(* IEC 61131-3 sources: volt/packages/volt-lsp-iec/test-corpus/lenze-mid/Device/Plc Logic/Application/Library Manager/(unresolved)/cmpopcuastack interfaces (part 3) *)

(* ---- OPCUA_NODEREFERENCE.dut ---- *)
TYPE OPCUA_NODEREFERENCE :
STRUCT
	NODEID : OpcUa_NodeId;
	REFERENCETYPEID : OpcUa_NodeId;
	ISFORWARD : OpcUa_Boolean;
	NOOFREFERENCEDNODEIDS : OpcUa_Int32;
	REFERENCEDNODEIDS : POINTER TO OpcUa_NodeId;
END_STRUCT
END_TYPE

(* ---- OPCUA_NODETYPEDESCRIPTION.dut ---- *)
TYPE OPCUA_NODETYPEDESCRIPTION :
STRUCT
	TYPEDEFINITIONNODE : OpcUa_ExpandedNodeId;
	INCLUDESUBTYPES : OpcUa_Boolean;
	NOOFDATATORETURN : OpcUa_Int32;
	DATATORETURN : POINTER TO OpcUa_QueryDataDescription;
END_STRUCT
END_TYPE

(* ---- OPCUA_NOTIFICATIONMESSAGE.dut ---- *)
TYPE OPCUA_NOTIFICATIONMESSAGE :
STRUCT
	SEQUENCENUMBER : OpcUa_UInt32;
	PUBLISHTIME : OpcUa_DateTime;
	NOOFNOTIFICATIONDATA : OpcUa_Int32;
	NOTIFICATIONDATA : POINTER TO OpcUa_ExtensionObject;
END_STRUCT
END_TYPE

(* ---- OPCUA_OBJECTATTRIBUTES.dut ---- *)
TYPE OPCUA_OBJECTATTRIBUTES :
STRUCT
	SPECIFIEDATTRIBUTES : OpcUa_UInt32;
	DISPLAYNAME : OpcUa_LocalizedText;
	DESCRIPTION : OpcUa_LocalizedText;
	WRITEMASK : OpcUa_UInt32;
	USERWRITEMASK : OpcUa_UInt32;
	EVENTNOTIFIER : OpcUa_Byte;
END_STRUCT
END_TYPE

(* ---- OPCUA_OBJECTTYPEATTRIBUTES.dut ---- *)
TYPE OPCUA_OBJECTTYPEATTRIBUTES :
STRUCT
	SPECIFIEDATTRIBUTES : OpcUa_UInt32;
	DISPLAYNAME : OpcUa_LocalizedText;
	DESCRIPTION : OpcUa_LocalizedText;
	WRITEMASK : OpcUa_UInt32;
	USERWRITEMASK : OpcUa_UInt32;
	ISABSTRACT : OpcUa_Boolean;
END_STRUCT
END_TYPE

(* ---- OPCUA_OPENSECURECHANNELREQUEST.dut ---- *)
TYPE OPCUA_OPENSECURECHANNELREQUEST :
STRUCT
	REQUESTHEADER : OpcUa_RequestHeader;
	CLIENTPROTOCOLVERSION : OpcUa_UInt32;
	REQUESTTYPE : OpcUa_SecurityTokenRequestType;
	SECURITYMODE : OpcUa_MessageSecurityMode;
	CLIENTNONCE : OpcUa_ByteString;
	REQUESTEDLIFETIME : OpcUa_UInt32;
END_STRUCT
END_TYPE

(* ---- OPCUA_OPENSECURECHANNELRESPONSE.dut ---- *)
TYPE OPCUA_OPENSECURECHANNELRESPONSE :
STRUCT
	RESPONSEHEADER : OpcUa_ResponseHeader;
	SERVERPROTOCOLVERSION : OpcUa_UInt32;
	SECURITYTOKEN : OpcUa_ChannelSecurityToken;
	SERVERNONCE : OpcUa_ByteString;
END_STRUCT
END_TYPE

(* ---- OPCUA_OPTIONSET.dut ---- *)
TYPE OPCUA_OPTIONSET :
STRUCT
	VALUE : OpcUa_ByteString;
	VALIDBITS : OpcUa_ByteString;
END_STRUCT
END_TYPE

(* ---- OPCUA_PARSINGRESULT.dut ---- *)
TYPE OPCUA_PARSINGRESULT :
STRUCT
	STATUSCODE : OpcUa_StatusCode;
	NOOFDATASTATUSCODES : OpcUa_Int32;
	DATASTATUSCODES : POINTER TO OpcUa_StatusCode;
	NOOFDATADIAGNOSTICINFOS : OpcUa_Int32;
	DATADIAGNOSTICINFOS : POINTER TO OpcUa_DiagnosticInfo;
END_STRUCT
END_TYPE

(* ---- OPCUA_PERFORMUPDATETYPE.dut ---- *)
TYPE OPCUA_PERFORMUPDATETYPE :
(
	OPCUA_PERFORMUPDATETYPE_INSERT := 1,
	OPCUA_PERFORMUPDATETYPE_REPLACE := 2,
	OPCUA_PERFORMUPDATETYPE_UPDATE := 3,
	OPCUA_PERFORMUPDATETYPE_REMOVE := 4
);
END_TYPE

(* ---- OPCUA_PROGRAMDIAGNOSTIC2DATATYPE.dut ---- *)
TYPE OPCUA_PROGRAMDIAGNOSTIC2DATATYPE :
STRUCT
	CREATESESSIONID : OpcUa_NodeId;
	CREATECLIENTNAME : OpcUa_String;
	INVOCATIONCREATIONTIME : OpcUa_DateTime;
	LASTTRANSITIONTIME : OpcUa_DateTime;
	LASTMETHODCALL : OpcUa_String;
	LASTMETHODSESSIONID : OpcUa_NodeId;
	NOOFLASTMETHODINPUTARGUMENTS : OpcUa_Int32;
	LASTMETHODINPUTARGUMENTS : POINTER TO OpcUa_Argument;
	NOOFLASTMETHODOUTPUTARGUMENTS : OpcUa_Int32;
	LASTMETHODOUTPUTARGUMENTS : POINTER TO OpcUa_Argument;
	NOOFLASTMETHODINPUTVALUES : OpcUa_Int32;
	LASTMETHODINPUTVALUES : POINTER TO OpcUa_Variant;
	NOOFLASTMETHODOUTPUTVALUES : OpcUa_Int32;
	LASTMETHODOUTPUTVALUES : POINTER TO OpcUa_Variant;
	LASTMETHODCALLTIME : OpcUa_DateTime;
	LASTMETHODRETURNSTATUS : OpcUa_StatusResult;
END_STRUCT
END_TYPE

(* ---- OPCUA_PROGRAMDIAGNOSTICDATATYPE.dut ---- *)
TYPE OPCUA_PROGRAMDIAGNOSTICDATATYPE :
STRUCT
	CREATESESSIONID : OpcUa_NodeId;
	CREATECLIENTNAME : OpcUa_String;
	INVOCATIONCREATIONTIME : OpcUa_DateTime;
	LASTTRANSITIONTIME : OpcUa_DateTime;
	LASTMETHODCALL : OpcUa_String;
	LASTMETHODSESSIONID : OpcUa_NodeId;
	NOOFLASTMETHODINPUTARGUMENTS : OpcUa_Int32;
	LASTMETHODINPUTARGUMENTS : POINTER TO OpcUa_Argument;
	NOOFLASTMETHODOUTPUTARGUMENTS : OpcUa_Int32;
	LASTMETHODOUTPUTARGUMENTS : POINTER TO OpcUa_Argument;
	LASTMETHODCALLTIME : OpcUa_DateTime;
	LASTMETHODRETURNSTATUS : OpcUa_StatusResult;
END_STRUCT
END_TYPE

(* ---- OPCUA_PUBLISHREQUEST.dut ---- *)
TYPE OPCUA_PUBLISHREQUEST :
STRUCT
	REQUESTHEADER : OpcUa_RequestHeader;
	NOOFSUBSCRIPTIONACKNOWLEDGEMENTS : OpcUa_Int32;
	SUBSCRIPTIONACKNOWLEDGEMENTS : POINTER TO OpcUa_SubscriptionAcknowledgement;
END_STRUCT
END_TYPE

(* ---- OPCUA_PUBLISHRESPONSE.dut ---- *)
TYPE OPCUA_PUBLISHRESPONSE :
STRUCT
	RESPONSEHEADER : OpcUa_ResponseHeader;
	SUBSCRIPTIONID : OpcUa_UInt32;
	NOOFAVAILABLESEQUENCENUMBERS : OpcUa_Int32;
	AVAILABLESEQUENCENUMBERS : POINTER TO OpcUa_UInt32;
	MORENOTIFICATIONS : OpcUa_Boolean;
	NOTIFICATIONMESSAGE : OpcUa_NotificationMessage;
	NOOFRESULTS : OpcUa_Int32;
	RESULTS : POINTER TO OpcUa_StatusCode;
	NOOFDIAGNOSTICINFOS : OpcUa_Int32;
	DIAGNOSTICINFOS : POINTER TO OpcUa_DiagnosticInfo;
END_STRUCT
END_TYPE

(* ---- OPCUA_QUALIFIEDNAME.dut ---- *)
TYPE OPCUA_QUALIFIEDNAME :
STRUCT
	NAMESPACEINDEX : OpcUa_UInt16;
	RESERVED : OpcUa_UInt16;
	NAME : OpcUa_String;
END_STRUCT
END_TYPE

(* ---- OPCUA_QUERYDATADESCRIPTION.dut ---- *)
TYPE OPCUA_QUERYDATADESCRIPTION :
STRUCT
	RELATIVEPATH : OpcUa_RelativePath;
	ATTRIBUTEID : OpcUa_UInt32;
	INDEXRANGE : OpcUa_String;
END_STRUCT
END_TYPE

(* ---- OPCUA_QUERYDATASET.dut ---- *)
TYPE OPCUA_QUERYDATASET :
STRUCT
	NODEID : OpcUa_ExpandedNodeId;
	TYPEDEFINITIONNODE : OpcUa_ExpandedNodeId;
	NOOFVALUES : OpcUa_Int32;
	VALUES : POINTER TO OpcUa_Variant;
END_STRUCT
END_TYPE

(* ---- OPCUA_QUERYFIRSTREQUEST.dut ---- *)
TYPE OPCUA_QUERYFIRSTREQUEST :
STRUCT
	REQUESTHEADER : OpcUa_RequestHeader;
	VIEW : OpcUa_ViewDescription;
	NOOFNODETYPES : OpcUa_Int32;
	NODETYPES : POINTER TO OpcUa_NodeTypeDescription;
	FILTER : OpcUa_ContentFilter;
	MAXDATASETSTORETURN : OpcUa_UInt32;
	MAXREFERENCESTORETURN : OpcUa_UInt32;
END_STRUCT
END_TYPE

(* ---- OPCUA_QUERYFIRSTRESPONSE.dut ---- *)
TYPE OPCUA_QUERYFIRSTRESPONSE :
STRUCT
	RESPONSEHEADER : OpcUa_ResponseHeader;
	NOOFQUERYDATASETS : OpcUa_Int32;
	QUERYDATASETS : POINTER TO OpcUa_QueryDataSet;
	CONTINUATIONPOINT : OpcUa_ByteString;
	NOOFPARSINGRESULTS : OpcUa_Int32;
	PARSINGRESULTS : POINTER TO OpcUa_ParsingResult;
	NOOFDIAGNOSTICINFOS : OpcUa_Int32;
	DIAGNOSTICINFOS : POINTER TO OpcUa_DiagnosticInfo;
	FILTERRESULT : OpcUa_ContentFilterResult;
END_STRUCT
END_TYPE

(* ---- OPCUA_QUERYNEXTREQUEST.dut ---- *)
TYPE OPCUA_QUERYNEXTREQUEST :
STRUCT
	REQUESTHEADER : OpcUa_RequestHeader;
	RELEASECONTINUATIONPOINT : OpcUa_Boolean;
	CONTINUATIONPOINT : OpcUa_ByteString;
END_STRUCT
END_TYPE

(* ---- OPCUA_QUERYNEXTRESPONSE.dut ---- *)
TYPE OPCUA_QUERYNEXTRESPONSE :
STRUCT
	RESPONSEHEADER : OpcUa_ResponseHeader;
	NOOFQUERYDATASETS : OpcUa_Int32;
	QUERYDATASETS : POINTER TO OpcUa_QueryDataSet;
	REVISEDCONTINUATIONPOINT : OpcUa_ByteString;
END_STRUCT
END_TYPE

(* ---- OPCUA_RANGE.dut ---- *)
TYPE OPCUA_RANGE :
STRUCT
	LOW : OpcUa_Double;
	HIGH : OpcUa_Double;
END_STRUCT
END_TYPE

(* ---- OPCUA_READATTIMEDETAILS.dut ---- *)
TYPE OPCUA_READATTIMEDETAILS :
STRUCT
	NOOFREQTIMES : OpcUa_Int32;
	REQTIMES : POINTER TO OpcUa_DateTime;
	USESIMPLEBOUNDS : OpcUa_Boolean;
END_STRUCT
END_TYPE

(* ---- OPCUA_READEVENTDETAILS.dut ---- *)
TYPE OPCUA_READEVENTDETAILS :
STRUCT
	NUMVALUESPERNODE : OpcUa_UInt32;
	STARTTIME : OpcUa_DateTime;
	ENDTIME : OpcUa_DateTime;
	FILTER : OpcUa_EventFilter;
END_STRUCT
END_TYPE

(* ---- OPCUA_READPROCESSEDDETAILS.dut ---- *)
TYPE OPCUA_READPROCESSEDDETAILS :
STRUCT
	STARTTIME : OpcUa_DateTime;
	ENDTIME : OpcUa_DateTime;
	PROCESSINGINTERVAL : OpcUa_Double;
	NOOFAGGREGATETYPE : OpcUa_Int32;
	AGGREGATETYPE : POINTER TO OpcUa_NodeId;
	AGGREGATECONFIGURATION : OpcUa_AggregateConfiguration;
END_STRUCT
END_TYPE

(* ---- OPCUA_READRAWMODIFIEDDETAILS.dut ---- *)
TYPE OPCUA_READRAWMODIFIEDDETAILS :
STRUCT
	ISREADMODIFIED : OpcUa_Boolean;
	STARTTIME : OpcUa_DateTime;
	ENDTIME : OpcUa_DateTime;
	NUMVALUESPERNODE : OpcUa_UInt32;
	RETURNBOUNDS : OpcUa_Boolean;
END_STRUCT
END_TYPE

(* ---- OPCUA_READREQUEST.dut ---- *)
TYPE OPCUA_READREQUEST :
STRUCT
	REQUESTHEADER : OpcUa_RequestHeader;
	MAXAGE : OpcUa_Double;
	TIMESTAMPSTORETURN : OpcUa_TimestampsToReturn;
	NOOFNODESTOREAD : OpcUa_Int32;
	NODESTOREAD : POINTER TO OpcUa_ReadValueId;
END_STRUCT
END_TYPE

(* ---- OPCUA_READRESPONSE.dut ---- *)
TYPE OPCUA_READRESPONSE :
STRUCT
	RESPONSEHEADER : OpcUa_ResponseHeader;
	NOOFRESULTS : OpcUa_Int32;
	RESULTS : POINTER TO OpcUa_DataValue;
	NOOFDIAGNOSTICINFOS : OpcUa_Int32;
	DIAGNOSTICINFOS : POINTER TO OpcUa_DiagnosticInfo;
END_STRUCT
END_TYPE

(* ---- OPCUA_READVALUEID.dut ---- *)
TYPE OPCUA_READVALUEID :
STRUCT
	NODEID : OpcUa_NodeId;
	ATTRIBUTEID : OpcUa_Attributes;
	INDEXRANGE : OpcUa_String;
	DATAENCODING : OpcUa_QualifiedName;
END_STRUCT
END_TYPE

(* ---- OPCUA_REDUNDANCYSUPPORT.dut ---- *)
TYPE OPCUA_REDUNDANCYSUPPORT :
(
	OPCUA_REDUNDANCYSUPPORT_NONE := 0,
	OPCUA_REDUNDANCYSUPPORT_COLD := 1,
	OPCUA_REDUNDANCYSUPPORT_WARM := 2,
	OPCUA_REDUNDANCYSUPPORT_HOT := 3,
	OPCUA_REDUNDANCYSUPPORT_TRANSPARENT := 4,
	OPCUA_REDUNDANCYSUPPORT_HOTANDMIRRORED := 5
);
END_TYPE

(* ---- OPCUA_REDUNDANTSERVERDATATYPE.dut ---- *)
TYPE OPCUA_REDUNDANTSERVERDATATYPE :
STRUCT
	SERVERID : OpcUa_String;
	SERVICELEVEL : OpcUa_Byte;
	SERVERSTATE : OpcUa_ServerState;
END_STRUCT
END_TYPE

(* ---- OPCUA_REFERENCEDESCRIPTION.dut ---- *)
TYPE OPCUA_REFERENCEDESCRIPTION :
STRUCT
	REFERENCETYPEID : OpcUa_NodeId;
	ISFORWARD : OpcUa_Boolean;
	NODEID : OpcUa_ExpandedNodeId;
	BROWSENAME : OpcUa_QualifiedName;
	DISPLAYNAME : OpcUa_LocalizedText;
	NODECLASS : OpcUa_NodeClass;
	TYPEDEFINITION : OpcUa_ExpandedNodeId;
END_STRUCT
END_TYPE

(* ---- OPCUA_REFERENCETYPEATTRIBUTES.dut ---- *)
TYPE OPCUA_REFERENCETYPEATTRIBUTES :
STRUCT
	SPECIFIEDATTRIBUTES : OpcUa_UInt32;
	DISPLAYNAME : OpcUa_LocalizedText;
	DESCRIPTION : OpcUa_LocalizedText;
	WRITEMASK : OpcUa_UInt32;
	USERWRITEMASK : OpcUa_UInt32;
	ISABSTRACT : OpcUa_Boolean;
	SYMMETRIC : OpcUa_Boolean;
	INVERSENAME : OpcUa_LocalizedText;
END_STRUCT
END_TYPE

(* ---- OPCUA_REGISTEREDSERVER.dut ---- *)
TYPE OPCUA_REGISTEREDSERVER :
STRUCT
	SERVERURI : OpcUa_String;
	PRODUCTURI : OpcUa_String;
	NOOFSERVERNAMES : OpcUa_Int32;
	SERVERNAMES : POINTER TO OpcUa_LocalizedText;
	SERVERTYPE : OpcUa_ApplicationType;
	GATEWAYSERVERURI : OpcUa_String;
	NOOFDISCOVERYURLS : OpcUa_Int32;
	DISCOVERYURLS : POINTER TO OpcUa_String;
	SEMAPHOREFILEPATH : OpcUa_String;
	ISONLINE : OpcUa_Boolean;
END_STRUCT
END_TYPE

(* ---- OPCUA_REGISTERNODESREQUEST.dut ---- *)
TYPE OPCUA_REGISTERNODESREQUEST :
STRUCT
	REQUESTHEADER : OpcUa_RequestHeader;
	NOOFNODESTOREGISTER : OpcUa_Int32;
	NODESTOREGISTER : POINTER TO OpcUa_NodeId;
END_STRUCT
END_TYPE

(* ---- OPCUA_REGISTERNODESRESPONSE.dut ---- *)
TYPE OPCUA_REGISTERNODESRESPONSE :
STRUCT
	RESPONSEHEADER : OpcUa_ResponseHeader;
	NOOFREGISTEREDNODEIDS : OpcUa_Int32;
	REGISTEREDNODEIDS : POINTER TO OpcUa_NodeId;
END_STRUCT
END_TYPE

(* ---- OPCUA_REGISTERSERVER2REQUEST.dut ---- *)
TYPE OPCUA_REGISTERSERVER2REQUEST :
STRUCT
	REQUESTHEADER : OpcUa_RequestHeader;
	SERVER : OpcUa_RegisteredServer;
	NOOFDISCOVERYCONFIGURATION : OpcUa_Int32;
	DISCOVERYCONFIGURATION : POINTER TO OpcUa_ExtensionObject;
END_STRUCT
END_TYPE

(* ---- OPCUA_REGISTERSERVER2RESPONSE.dut ---- *)
TYPE OPCUA_REGISTERSERVER2RESPONSE :
STRUCT
	RESPONSEHEADER : OpcUa_ResponseHeader;
	NOOFCONFIGURATIONRESULTS : OpcUa_Int32;
	CONFIGURATIONRESULTS : POINTER TO OpcUa_StatusCode;
	NOOFDIAGNOSTICINFOS : OpcUa_Int32;
	DIAGNOSTICINFOS : POINTER TO OpcUa_DiagnosticInfo;
END_STRUCT
END_TYPE

(* ---- OPCUA_REGISTERSERVERREQUEST.dut ---- *)
TYPE OPCUA_REGISTERSERVERREQUEST :
STRUCT
	REQUESTHEADER : OpcUa_RequestHeader;
	SERVER : OpcUa_RegisteredServer;
END_STRUCT
END_TYPE

(* ---- OPCUA_REGISTERSERVERRESPONSE.dut ---- *)
TYPE OPCUA_REGISTERSERVERRESPONSE :
STRUCT
	RESPONSEHEADER : OpcUa_ResponseHeader;
END_STRUCT
END_TYPE

(* ---- OPCUA_RELATIVEPATH.dut ---- *)
TYPE OPCUA_RELATIVEPATH :
STRUCT
	NOOFELEMENTS : OpcUa_Int32;
	ELEMENTS : POINTER TO OpcUa_RelativePathElement;
END_STRUCT
END_TYPE

(* ---- OPCUA_RELATIVEPATHELEMENT.dut ---- *)
TYPE OPCUA_RELATIVEPATHELEMENT :
STRUCT
	REFERENCETYPEID : OpcUa_NodeId;
	ISINVERSE : OpcUa_Boolean;
	INCLUDESUBTYPES : OpcUa_Boolean;
	TARGETNAME : OpcUa_QualifiedName;
END_STRUCT
END_TYPE

(* ---- OPCUA_REPUBLISHREQUEST.dut ---- *)
TYPE OPCUA_REPUBLISHREQUEST :
STRUCT
	REQUESTHEADER : OpcUa_RequestHeader;
	SUBSCRIPTIONID : OpcUa_UInt32;
	RETRANSMITSEQUENCENUMBER : OpcUa_UInt32;
END_STRUCT
END_TYPE

(* ---- OPCUA_REPUBLISHRESPONSE.dut ---- *)
TYPE OPCUA_REPUBLISHRESPONSE :
STRUCT
	RESPONSEHEADER : OpcUa_ResponseHeader;
	NOTIFICATIONMESSAGE : OpcUa_NotificationMessage;
END_STRUCT
END_TYPE

(* ---- OPCUA_REQUESTHEADER.dut ---- *)
TYPE OPCUA_REQUESTHEADER :
STRUCT
	AUTHENTICATIONTOKEN : OpcUa_NodeId;
	TIMESTAMP : OpcUa_DateTime;
	REQUESTHANDLE : OpcUa_UInt32;
	RETURNDIAGNOSTICS : OpcUa_UInt32;
	AUDITENTRYID : OpcUa_String;
	TIMEOUTHINT : OpcUa_UInt32;
	ADDITIONALHEADER : OpcUa_ExtensionObject;
END_STRUCT
END_TYPE

(* ---- OPCUA_RESPONSEHEADER.dut ---- *)
TYPE OPCUA_RESPONSEHEADER :
STRUCT
	TIMESTAMP : OpcUa_DateTime;
	REQUESTHANDLE : OpcUa_UInt32;
	SERVICERESULT : OpcUa_StatusCode;
	SERVICEDIAGNOSTICS : OpcUa_DiagnosticInfo;
	NOOFSTRINGTABLE : OpcUa_Int32;
	STRINGTABLE : POINTER TO OpcUa_String;
	ADDITIONALHEADER : OpcUa_ExtensionObject;
END_STRUCT
END_TYPE

(* ---- OPCUA_ROLEPERMISSIONTYPE.dut ---- *)
TYPE OPCUA_ROLEPERMISSIONTYPE :
STRUCT
	ROLEID : OpcUa_NodeId;
	PERMISSIONS : OpcUa_UInt32;
END_STRUCT
END_TYPE

(* ---- OPCUA_SAMPLINGINTERVALDIAGNOSTICSDATATYPE.dut ---- *)
TYPE OPCUA_SAMPLINGINTERVALDIAGNOSTICSDATATYPE :
STRUCT
	SAMPLINGINTERVAL : OpcUa_Double;
	MONITOREDITEMCOUNT : OpcUa_UInt32;
	MAXMONITOREDITEMCOUNT : OpcUa_UInt32;
	DISABLEDMONITOREDITEMCOUNT : OpcUa_UInt32;
END_STRUCT
END_TYPE

(* ---- OPCUA_SBYTE.dut ---- *)
TYPE OPCUA_SBYTE : SINT;
END_TYPE

(* ---- OPCUA_SECURITYTOKENREQUESTTYPE.dut ---- *)
TYPE OPCUA_SECURITYTOKENREQUESTTYPE :
(
	OPCUA_SECURITYTOKENREQUESTTYPE_ISSUE := 0,
	OPCUA_SECURITYTOKENREQUESTTYPE_RENEW := 1
);
END_TYPE

(* ---- OPCUA_SEMANTICCHANGESTRUCTUREDATATYPE.dut ---- *)
TYPE OPCUA_SEMANTICCHANGESTRUCTUREDATATYPE :
STRUCT
	AFFECTED : OpcUa_NodeId;
	AFFECTEDTYPE : OpcUa_NodeId;
END_STRUCT
END_TYPE

(* ---- OPCUA_SERVERDIAGNOSTICSSUMMARYDATATYPE.dut ---- *)
TYPE OPCUA_SERVERDIAGNOSTICSSUMMARYDATATYPE :
STRUCT
	SERVERVIEWCOUNT : OpcUa_UInt32;
	CURRENTSESSIONCOUNT : OpcUa_UInt32;
	CUMULATEDSESSIONCOUNT : OpcUa_UInt32;
	SECURITYREJECTEDSESSIONCOUNT : OpcUa_UInt32;
	REJECTEDSESSIONCOUNT : OpcUa_UInt32;
	SESSIONTIMEOUTCOUNT : OpcUa_UInt32;
	SESSIONABORTCOUNT : OpcUa_UInt32;
	CURRENTSUBSCRIPTIONCOUNT : OpcUa_UInt32;
	CUMULATEDSUBSCRIPTIONCOUNT : OpcUa_UInt32;
	PUBLISHINGINTERVALCOUNT : OpcUa_UInt32;
	SECURITYREJECTEDREQUESTSCOUNT : OpcUa_UInt32;
	REJECTEDREQUESTSCOUNT : OpcUa_UInt32;
END_STRUCT
END_TYPE

(* ---- OPCUA_SERVERONNETWORK.dut ---- *)
TYPE OPCUA_SERVERONNETWORK :
STRUCT
	RECORDID : OpcUa_UInt32;
	SERVERNAME : OpcUa_String;
	DISCOVERYURL : OpcUa_String;
	NOOFSERVERCAPABILITIES : OpcUa_Int32;
	SERVERCAPABILITIES : POINTER TO OpcUa_String;
END_STRUCT
END_TYPE

(* ---- OPCUA_SERVERSTATE.dut ---- *)
TYPE OPCUA_SERVERSTATE :
(
	OPCUA_SERVERSTATE_RUNNING := 0,
	OPCUA_SERVERSTATE_FAILED := 1,
	OPCUA_SERVERSTATE_NOCONFIGURATION := 2,
	OPCUA_SERVERSTATE_SUSPENDED := 3,
	OPCUA_SERVERSTATE_SHUTDOWN := 4,
	OPCUA_SERVERSTATE_TEST := 5,
	OPCUA_SERVERSTATE_COMMUNICATIONFAULT := 6,
	OPCUA_SERVERSTATE_UNKNOWN := 7
);
END_TYPE

(* ---- OPCUA_SERVERSTATUSDATATYPE.dut ---- *)
TYPE OPCUA_SERVERSTATUSDATATYPE :
STRUCT
	STARTTIME : OpcUa_DateTime;
	CURRENTTIME : OpcUa_DateTime;
	STATE : OpcUa_ServerState;
	BUILDINFO : OpcUa_BuildInfo;
	SECONDSTILLSHUTDOWN : OpcUa_UInt32;
	SHUTDOWNREASON : OpcUa_LocalizedText;
END_STRUCT
END_TYPE

(* ---- OPCUA_SERVICECOUNTERDATATYPE.dut ---- *)
TYPE OPCUA_SERVICECOUNTERDATATYPE :
STRUCT
	TOTALCOUNT : OpcUa_UInt32;
	ERRORCOUNT : OpcUa_UInt32;
END_STRUCT
END_TYPE

(* ---- OPCUA_SERVICEFAULT.dut ---- *)
TYPE OPCUA_SERVICEFAULT :
STRUCT
	RESPONSEHEADER : OpcUa_ResponseHeader;
END_STRUCT
END_TYPE

(* ---- OPCUA_SESSIONDIAGNOSTICSDATATYPE.dut ---- *)
TYPE OPCUA_SESSIONDIAGNOSTICSDATATYPE :
STRUCT
	SESSIONID : OpcUa_NodeId;
	SESSIONNAME : OpcUa_String;
	CLIENTDESCRIPTION : OpcUa_ApplicationDescription;
	SERVERURI : OpcUa_String;
	ENDPOINTURL : OpcUa_String;
	NOOFLOCALEIDS : OpcUa_Int32;
	LOCALEIDS : POINTER TO OpcUa_String;
	ACTUALSESSIONTIMEOUT : OpcUa_Double;
	MAXRESPONSEMESSAGESIZE : OpcUa_UInt32;
	CLIENTCONNECTIONTIME : OpcUa_DateTime;
	CLIENTLASTCONTACTTIME : OpcUa_DateTime;
	CURRENTSUBSCRIPTIONSCOUNT : OpcUa_UInt32;
	CURRENTMONITOREDITEMSCOUNT : OpcUa_UInt32;
	CURRENTPUBLISHREQUESTSINQUEUE : OpcUa_UInt32;
	TOTALREQUESTCOUNT : OpcUa_ServiceCounterDataType;
	UNAUTHORIZEDREQUESTCOUNT : OpcUa_UInt32;
	READCOUNT : OpcUa_ServiceCounterDataType;
	HISTORYREADCOUNT : OpcUa_ServiceCounterDataType;
	WRITECOUNT : OpcUa_ServiceCounterDataType;
	HISTORYUPDATECOUNT : OpcUa_ServiceCounterDataType;
	CALLCOUNT : OpcUa_ServiceCounterDataType;
	CREATEMONITOREDITEMSCOUNT : OpcUa_ServiceCounterDataType;
	MODIFYMONITOREDITEMSCOUNT : OpcUa_ServiceCounterDataType;
	SETMONITORINGMODECOUNT : OpcUa_ServiceCounterDataType;
	SETTRIGGERINGCOUNT : OpcUa_ServiceCounterDataType;
	DELETEMONITOREDITEMSCOUNT : OpcUa_ServiceCounterDataType;
	CREATESUBSCRIPTIONCOUNT : OpcUa_ServiceCounterDataType;
	MODIFYSUBSCRIPTIONCOUNT : OpcUa_ServiceCounterDataType;
	SETPUBLISHINGMODECOUNT : OpcUa_ServiceCounterDataType;
	PUBLISHCOUNT : OpcUa_ServiceCounterDataType;
	REPUBLISHCOUNT : OpcUa_ServiceCounterDataType;
	TRANSFERSUBSCRIPTIONSCOUNT : OpcUa_ServiceCounterDataType;
	DELETESUBSCRIPTIONSCOUNT : OpcUa_ServiceCounterDataType;
	ADDNODESCOUNT : OpcUa_ServiceCounterDataType;
	ADDREFERENCESCOUNT : OpcUa_ServiceCounterDataType;
	DELETENODESCOUNT : OpcUa_ServiceCounterDataType;
	DELETEREFERENCESCOUNT : OpcUa_ServiceCounterDataType;
	BROWSECOUNT : OpcUa_ServiceCounterDataType;
	BROWSENEXTCOUNT : OpcUa_ServiceCounterDataType;
	TRANSLATEBROWSEPATHSTONODEIDSCOUNT : OpcUa_ServiceCounterDataType;
	QUERYFIRSTCOUNT : OpcUa_ServiceCounterDataType;
	QUERYNEXTCOUNT : OpcUa_ServiceCounterDataType;
	REGISTERNODESCOUNT : OpcUa_ServiceCounterDataType;
	UNREGISTERNODESCOUNT : OpcUa_ServiceCounterDataType;
END_STRUCT
END_TYPE

(* ---- OPCUA_SESSIONLESSINVOKEREQUESTTYPE.dut ---- *)
TYPE OPCUA_SESSIONLESSINVOKEREQUESTTYPE :
STRUCT
	NOOFURISVERSION : OpcUa_Int32;
	URISVERSION : POINTER TO OpcUa_UInt32;
	NOOFNAMESPACEURIS : OpcUa_Int32;
	NAMESPACEURIS : POINTER TO OpcUa_String;
	NOOFSERVERURIS : OpcUa_Int32;
	SERVERURIS : POINTER TO OpcUa_String;
	NOOFLOCALEIDS : OpcUa_Int32;
	LOCALEIDS : POINTER TO OpcUa_String;
	SERVICEID : OpcUa_UInt32;
END_STRUCT
END_TYPE

(* ---- OPCUA_SESSIONLESSINVOKERESPONSETYPE.dut ---- *)
TYPE OPCUA_SESSIONLESSINVOKERESPONSETYPE :
STRUCT
	NOOFNAMESPACEURIS : OpcUa_Int32;
	NAMESPACEURIS : POINTER TO OpcUa_String;
	NOOFSERVERURIS : OpcUa_Int32;
	SERVERURIS : POINTER TO OpcUa_String;
	SERVICEID : OpcUa_UInt32;
END_STRUCT
END_TYPE

(* ---- OPCUA_SESSIONSECURITYDIAGNOSTICSDATATYPE.dut ---- *)
TYPE OPCUA_SESSIONSECURITYDIAGNOSTICSDATATYPE :
STRUCT
	SESSIONID : OpcUa_NodeId;
	CLIENTUSERIDOFSESSION : OpcUa_String;
	NOOFCLIENTUSERIDHISTORY : OpcUa_Int32;
	CLIENTUSERIDHISTORY : POINTER TO OpcUa_String;
	AUTHENTICATIONMECHANISM : OpcUa_String;
	ENCODING : OpcUa_String;
	TRANSPORTPROTOCOL : OpcUa_String;
	SECURITYMODE : OpcUa_MessageSecurityMode;
	SECURITYPOLICYURI : OpcUa_String;
	CLIENTCERTIFICATE : OpcUa_ByteString;
END_STRUCT
END_TYPE

(* ---- OPCUA_SETMONITORINGMODEREQUEST.dut ---- *)
TYPE OPCUA_SETMONITORINGMODEREQUEST :
STRUCT
	REQUESTHEADER : OpcUa_RequestHeader;
	SUBSCRIPTIONID : OpcUa_UInt32;
	MONITORINGMODE : OpcUa_MonitoringMode;
	NOOFMONITOREDITEMIDS : OpcUa_Int32;
	MONITOREDITEMIDS : POINTER TO OpcUa_UInt32;
END_STRUCT
END_TYPE

(* ---- OPCUA_SETMONITORINGMODERESPONSE.dut ---- *)
TYPE OPCUA_SETMONITORINGMODERESPONSE :
STRUCT
	RESPONSEHEADER : OpcUa_ResponseHeader;
	NOOFRESULTS : OpcUa_Int32;
	RESULTS : POINTER TO OpcUa_StatusCode;
	NOOFDIAGNOSTICINFOS : OpcUa_Int32;
	DIAGNOSTICINFOS : POINTER TO OpcUa_DiagnosticInfo;
END_STRUCT
END_TYPE

(* ---- OPCUA_SETPUBLISHINGMODEREQUEST.dut ---- *)
TYPE OPCUA_SETPUBLISHINGMODEREQUEST :
STRUCT
	REQUESTHEADER : OpcUa_RequestHeader;
	PUBLISHINGENABLED : OpcUa_Boolean;
	NOOFSUBSCRIPTIONIDS : OpcUa_Int32;
	SUBSCRIPTIONIDS : POINTER TO OpcUa_UInt32;
END_STRUCT
END_TYPE

(* ---- OPCUA_SETPUBLISHINGMODERESPONSE.dut ---- *)
TYPE OPCUA_SETPUBLISHINGMODERESPONSE :
STRUCT
	RESPONSEHEADER : OpcUa_ResponseHeader;
	NOOFRESULTS : OpcUa_Int32;
	RESULTS : POINTER TO OpcUa_StatusCode;
	NOOFDIAGNOSTICINFOS : OpcUa_Int32;
	DIAGNOSTICINFOS : POINTER TO OpcUa_DiagnosticInfo;
END_STRUCT
END_TYPE

(* ---- OPCUA_SETTRIGGERINGREQUEST.dut ---- *)
TYPE OPCUA_SETTRIGGERINGREQUEST :
STRUCT
	REQUESTHEADER : OpcUa_RequestHeader;
	SUBSCRIPTIONID : OpcUa_UInt32;
	TRIGGERINGITEMID : OpcUa_UInt32;
	NOOFLINKSTOADD : OpcUa_Int32;
	LINKSTOADD : POINTER TO OpcUa_UInt32;
	NOOFLINKSTOREMOVE : OpcUa_Int32;
	LINKSTOREMOVE : POINTER TO OpcUa_UInt32;
END_STRUCT
END_TYPE

(* ---- OPCUA_SETTRIGGERINGRESPONSE.dut ---- *)
TYPE OPCUA_SETTRIGGERINGRESPONSE :
STRUCT
	RESPONSEHEADER : OpcUa_ResponseHeader;
	NOOFADDRESULTS : OpcUa_Int32;
	ADDRESULTS : POINTER TO OpcUa_StatusCode;
	NOOFADDDIAGNOSTICINFOS : OpcUa_Int32;
	ADDDIAGNOSTICINFOS : POINTER TO OpcUa_DiagnosticInfo;
	NOOFREMOVERESULTS : OpcUa_Int32;
	REMOVERESULTS : POINTER TO OpcUa_StatusCode;
	NOOFREMOVEDIAGNOSTICINFOS : OpcUa_Int32;
	REMOVEDIAGNOSTICINFOS : POINTER TO OpcUa_DiagnosticInfo;
END_STRUCT
END_TYPE

(* ---- OPCUA_SIGNATUREDATA.dut ---- *)
TYPE OPCUA_SIGNATUREDATA :
STRUCT
	ALGORITHM : OpcUa_String;
	SIGNATURE : OpcUa_ByteString;
END_STRUCT
END_TYPE

(* ---- OPCUA_SIGNEDSOFTWARECERTIFICATE.dut ---- *)
TYPE OPCUA_SIGNEDSOFTWARECERTIFICATE :
STRUCT
	CERTIFICATEDATA : OpcUa_ByteString;
	SIGNATURE : OpcUa_ByteString;
END_STRUCT
END_TYPE

(* ---- OPCUA_SIMPLEATTRIBUTEOPERAND.dut ---- *)
TYPE OPCUA_SIMPLEATTRIBUTEOPERAND :
STRUCT
	TYPEDEFINITIONID : OpcUa_NodeId;
	NOOFBROWSEPATH : OpcUa_Int32;
	BROWSEPATH : POINTER TO OpcUa_QualifiedName;
	ATTRIBUTEID : OpcUa_UInt32;
	INDEXRANGE : OpcUa_String;
END_STRUCT
END_TYPE

(* ---- OPCUA_STATUSCHANGENOTIFICATION.dut ---- *)
TYPE OPCUA_STATUSCHANGENOTIFICATION :
STRUCT
	STATUS : OpcUa_StatusCode;
	DIAGNOSTICINFO : OpcUa_DiagnosticInfo;
END_STRUCT
END_TYPE

(* ---- OPCUA_STATUSCODE.dut ---- *)
TYPE OPCUA_STATUSCODE :
(
	OPCUA_GOOD := 0,
	OPCUA_BADUNEXPECTEDERROR := 16#80010000,
	OPCUA_BADINTERNALERROR := 16#80020000,
	OPCUA_BADOUTOFMEMORY := 16#80030000,
	OPCUA_BADRESOURCEUNAVAILABLE := 16#80040000,
	OPCUA_BADCOMMUNICATIONERROR := 16#80050000,
	OPCUA_BADENCODINGERROR := 16#80060000,
	OPCUA_BADDECODINGERROR := 16#80070000,
	OPCUA_BADENCODINGLIMITSEXCEEDED := 16#80080000,
	OPCUA_BADREQUESTTOOLARGE := 16#80B80000,
	OPCUA_BADRESPONSETOOLARGE := 16#80B90000,
	OPCUA_BADUNKNOWNRESPONSE := 16#80090000,
	OPCUA_BADTIMEOUT := 16#800A0000,
	OPCUA_BADSERVICEUNSUPPORTED := 16#800B0000,
	OPCUA_BADSHUTDOWN := 16#800C0000,
	OPCUA_BADSERVERNOTCONNECTED := 16#800D0000,
	OPCUA_BADSERVERHALTED := 16#800E0000,
	OPCUA_BADNOTHINGTODO := 16#800F0000,
	OPCUA_BADTOOMANYOPERATIONS := 16#80100000,
	OPCUA_BADTOOMANYMONITOREDITEMS := 16#80DB0000,
	OPCUA_BADDATATYPEIDUNKNOWN := 16#80110000,
	OPCUA_BADCERTIFICATEINVALID := 16#80120000,
	OPCUA_BADSECURITYCHECKSFAILED := 16#80130000,
	OPCUA_BADCERTIFICATEPOLICYCHECKFAILED := 16#81140000,
	OPCUA_BADCERTIFICATETIMEINVALID := 16#80140000,
	OPCUA_BADCERTIFICATEISSUERTIMEINVALID := 16#80150000,
	OPCUA_BADCERTIFICATEHOSTNAMEINVALID := 16#80160000,
	OPCUA_BADCERTIFICATEURIINVALID := 16#80170000,
	OPCUA_BADCERTIFICATEUSENOTALLOWED := 16#80180000,
	OPCUA_BADCERTIFICATEISSUERUSENOTALLOWED := 16#80190000,
	OPCUA_BADCERTIFICATEUNTRUSTED := 16#801A0000,
	OPCUA_BADCERTIFICATEREVOCATIONUNKNOWN := 16#801B0000,
	OPCUA_BADCERTIFICATEISSUERREVOCATIONUNKNOWN := 16#801C0000,
	OPCUA_BADCERTIFICATEREVOKED := 16#801D0000,
	OPCUA_BADCERTIFICATEISSUERREVOKED := 16#801E0000,
	OPCUA_BADCERTIFICATECHAININCOMPLETE := 16#810D0000,
	OPCUA_BADUSERACCESSDENIED := 16#801F0000,
	OPCUA_BADIDENTITYTOKENINVALID := 16#80200000,
	OPCUA_BADIDENTITYTOKENREJECTED := 16#80210000,
	OPCUA_BADSECURECHANNELIDINVALID := 16#80220000,
	OPCUA_BADINVALIDTIMESTAMP := 16#80230000,
	OPCUA_BADNONCEINVALID := 16#80240000,
	OPCUA_BADSESSIONIDINVALID := 16#80250000,
	OPCUA_BADSESSIONCLOSED := 16#80260000,
	OPCUA_BADSESSIONNOTACTIVATED := 16#80270000,
	OPCUA_BADSUBSCRIPTIONIDINVALID := 16#80280000,
	OPCUA_BADREQUESTHEADERINVALID := 16#802A0000,
	OPCUA_BADTIMESTAMPSTORETURNINVALID := 16#802B0000,
	OPCUA_BADREQUESTCANCELLEDBYCLIENT := 16#802C0000,
	OPCUA_BADTOOMANYARGUMENTS := 16#80E50000,
	OPCUA_BADLICENSEEXPIRED := 16#810E0000,
	OPCUA_BADLICENSELIMITSEXCEEDED := 16#810F0000,
	OPCUA_BADLICENSENOTAVAILABLE := 16#81100000,
	OPCUA_GOODSUBSCRIPTIONTRANSFERRED := 16#2D0000,
	OPCUA_GOODCOMPLETESASYNCHRONOUSLY := 16#2E0000,
	OPCUA_GOODOVERLOAD := 16#2F0000,
	OPCUA_GOODCLAMPED := 16#300000,
	OPCUA_BADNOCOMMUNICATION := 16#80310000,
	OPCUA_BADWAITINGFORINITIALDATA := 16#80320000,
	OPCUA_BADNODEIDINVALID := 16#80330000,
	OPCUA_BADNODEIDUNKNOWN := 16#80340000,
	OPCUA_BADATTRIBUTEIDINVALID := 16#80350000,
	OPCUA_BADINDEXRANGEINVALID := 16#80360000,
	OPCUA_BADINDEXRANGENODATA := 16#80370000,
	OPCUA_BADDATAENCODINGINVALID := 16#80380000,
	OPCUA_BADDATAENCODINGUNSUPPORTED := 16#80390000,
	OPCUA_BADNOTREADABLE := 16#803A0000,
	OPCUA_BADNOTWRITABLE := 16#803B0000,
	OPCUA_BADOUTOFRANGE := 16#803C0000,
	OPCUA_BADNOTSUPPORTED := 16#803D0000,
	OPCUA_BADNOTFOUND := 16#803E0000,
	OPCUA_BADOBJECTDELETED := 16#803F0000,
	OPCUA_BADNOTIMPLEMENTED := 16#80400000,
	OPCUA_BADMONITORINGMODEINVALID := 16#80410000,
	OPCUA_BADMONITOREDITEMIDINVALID := 16#80420000,
	OPCUA_BADMONITOREDITEMFILTERINVALID := 16#80430000,
	OPCUA_BADMONITOREDITEMFILTERUNSUPPORTED := 16#80440000,
	OPCUA_BADFILTERNOTALLOWED := 16#80450000,
	OPCUA_BADSTRUCTUREMISSING := 16#80460000,
	OPCUA_BADEVENTFILTERINVALID := 16#80470000,
	OPCUA_BADCONTENTFILTERINVALID := 16#80480000,
	OPCUA_BADFILTEROPERATORINVALID := 16#80C10000,
	OPCUA_BADFILTEROPERATORUNSUPPORTED := 16#80C20000,
	OPCUA_BADFILTEROPERANDCOUNTMISMATCH := 16#80C30000,
	OPCUA_BADFILTEROPERANDINVALID := 16#80490000,
	OPCUA_BADFILTERELEMENTINVALID := 16#80C40000,
	OPCUA_BADFILTERLITERALINVALID := 16#80C50000,
	OPCUA_BADCONTINUATIONPOINTINVALID := 16#804A0000,
	OPCUA_BADNOCONTINUATIONPOINTS := 16#804B0000,
	OPCUA_BADREFERENCETYPEIDINVALID := 16#804C0000,
	OPCUA_BADBROWSEDIRECTIONINVALID := 16#804D0000,
	OPCUA_BADNODENOTINVIEW := 16#804E0000,
	OPCUA_BADNUMERICOVERFLOW := 16#81120000,
	OPCUA_BADSERVERURIINVALID := 16#804F0000,
	OPCUA_BADSERVERNAMEMISSING := 16#80500000,
	OPCUA_BADDISCOVERYURLMISSING := 16#80510000,
	OPCUA_BADSEMPAHOREFILEMISSING := 16#80520000,
	OPCUA_BADREQUESTTYPEINVALID := 16#80530000,
	OPCUA_BADSECURITYMODEREJECTED := 16#80540000,
	OPCUA_BADSECURITYPOLICYREJECTED := 16#80550000,
	OPCUA_BADTOOMANYSESSIONS := 16#80560000,
	OPCUA_BADUSERSIGNATUREINVALID := 16#80570000,
	OPCUA_BADAPPLICATIONSIGNATUREINVALID := 16#80580000,
	OPCUA_BADNOVALIDCERTIFICATES := 16#80590000,
	OPCUA_BADIDENTITYCHANGENOTSUPPORTED := 16#80C60000,
	OPCUA_BADREQUESTCANCELLEDBYREQUEST := 16#805A0000,
	OPCUA_BADPARENTNODEIDINVALID := 16#805B0000,
	OPCUA_BADREFERENCENOTALLOWED := 16#805C0000,
	OPCUA_BADNODEIDREJECTED := 16#805D0000,
	OPCUA_BADNODEIDEXISTS := 16#805E0000,
	OPCUA_BADNODECLASSINVALID := 16#805F0000,
	OPCUA_BADBROWSENAMEINVALID := 16#80600000,
	OPCUA_BADBROWSENAMEDUPLICATED := 16#80610000,
	OPCUA_BADNODEATTRIBUTESINVALID := 16#80620000,
	OPCUA_BADTYPEDEFINITIONINVALID := 16#80630000,
	OPCUA_BADSOURCENODEIDINVALID := 16#80640000,
	OPCUA_BADTARGETNODEIDINVALID := 16#80650000,
	OPCUA_BADDUPLICATEREFERENCENOTALLOWED := 16#80660000,
	OPCUA_BADINVALIDSELFREFERENCE := 16#80670000,
	OPCUA_BADREFERENCELOCALONLY := 16#80680000,
	OPCUA_BADNODELETERIGHTS := 16#80690000,
	OPCUA_UNCERTAINREFERENCENOTDELETED := 16#40BC0000,
	OPCUA_BADSERVERINDEXINVALID := 16#806A0000,
	OPCUA_BADVIEWIDUNKNOWN := 16#806B0000,
	OPCUA_BADVIEWTIMESTAMPINVALID := 16#80C90000,
	OPCUA_BADVIEWPARAMETERMISMATCH := 16#80CA0000,
	OPCUA_BADVIEWVERSIONINVALID := 16#80CB0000,
	OPCUA_UNCERTAINNOTALLNODESAVAILABLE := 16#40C00000,
	OPCUA_GOODRESULTSMAYBEINCOMPLETE := 16#BA0000,
	OPCUA_BADNOTTYPEDEFINITION := 16#80C80000,
	OPCUA_UNCERTAINREFERENCEOUTOFSERVER := 16#406C0000,
	OPCUA_BADTOOMANYMATCHES := 16#806D0000,
	OPCUA_BADQUERYTOOCOMPLEX := 16#806E0000,
	OPCUA_BADNOMATCH := 16#806F0000,
	OPCUA_BADMAXAGEINVALID := 16#80700000,
	OPCUA_BADSECURITYMODEINSUFFICIENT := 16#80E60000,
	OPCUA_BADHISTORYOPERATIONINVALID := 16#80710000,
	OPCUA_BADHISTORYOPERATIONUNSUPPORTED := 16#80720000,
	OPCUA_BADINVALIDTIMESTAMPARGUMENT := 16#80BD0000,
	OPCUA_BADWRITENOTSUPPORTED := 16#80730000,
	OPCUA_BADTYPEMISMATCH := 16#80740000,
	OPCUA_BADMETHODINVALID := 16#80750000,
	OPCUA_BADARGUMENTSMISSING := 16#80760000,
	OPCUA_BADNOTEXECUTABLE := 16#81110000,
	OPCUA_BADTOOMANYSUBSCRIPTIONS := 16#80770000,
	OPCUA_BADTOOMANYPUBLISHREQUESTS := 16#80780000,
	OPCUA_BADNOSUBSCRIPTION := 16#80790000,
	OPCUA_BADSEQUENCENUMBERUNKNOWN := 16#807A0000,
	OPCUA_BADMESSAGENOTAVAILABLE := 16#807B0000,
	OPCUA_BADINSUFFICIENTCLIENTPROFILE := 16#807C0000,
	OPCUA_BADSTATENOTACTIVE := 16#80BF0000,
	OPCUA_BADALREADYEXISTS := 16#81150000,
	OPCUA_BADTCPSERVERTOOBUSY := 16#807D0000,
	OPCUA_BADTCPMESSAGETYPEINVALID := 16#807E0000,
	OPCUA_BADTCPSECURECHANNELUNKNOWN := 16#807F0000,
	OPCUA_BADTCPMESSAGETOOLARGE := 16#80800000,
	OPCUA_BADTCPNOTENOUGHRESOURCES := 16#80810000,
	OPCUA_BADTCPINTERNALERROR := 16#80820000,
	OPCUA_BADTCPENDPOINTURLINVALID := 16#80830000,
	OPCUA_BADREQUESTINTERRUPTED := 16#80840000,
	OPCUA_BADREQUESTTIMEOUT := 16#80850000,
	OPCUA_BADSECURECHANNELCLOSED := 16#80860000,
	OPCUA_BADSECURECHANNELTOKENUNKNOWN := 16#80870000,
	OPCUA_BADSEQUENCENUMBERINVALID := 16#80880000,
	OPCUA_BADPROTOCOLVERSIONUNSUPPORTED := 16#80BE0000,
	OPCUA_BADCONFIGURATIONERROR := 16#80890000,
	OPCUA_BADNOTCONNECTED := 16#808A0000,
	OPCUA_BADDEVICEFAILURE := 16#808B0000,
	OPCUA_BADSENSORFAILURE := 16#808C0000,
	OPCUA_BADOUTOFSERVICE := 16#808D0000,
	OPCUA_BADDEADBANDFILTERINVALID := 16#808E0000,
	OPCUA_UNCERTAINNOCOMMUNICATIONLASTUSABLEVALUE := 16#408F0000,
	OPCUA_UNCERTAINLASTUSABLEVALUE := 16#40900000,
	OPCUA_UNCERTAINSUBSTITUTEVALUE := 16#40910000,
	OPCUA_UNCERTAININITIALVALUE := 16#40920000,
	OPCUA_UNCERTAINSENSORNOTACCURATE := 16#40930000,
	OPCUA_UNCERTAINENGINEERINGUNITSEXCEEDED := 16#40940000,
	OPCUA_UNCERTAINSUBNORMAL := 16#40950000,
	OPCUA_GOODLOCALOVERRIDE := 16#960000,
	OPCUA_BADREFRESHINPROGRESS := 16#80970000,
	OPCUA_BADCONDITIONALREADYDISABLED := 16#80980000,
	OPCUA_BADCONDITIONALREADYENABLED := 16#80CC0000,
	OPCUA_BADCONDITIONDISABLED := 16#80990000,
	OPCUA_BADEVENTIDUNKNOWN := 16#809A0000,
	OPCUA_BADEVENTNOTACKNOWLEDGEABLE := 16#80BB0000,
	OPCUA_BADDIALOGNOTACTIVE := 16#80CD0000,
	OPCUA_BADDIALOGRESPONSEINVALID := 16#80CE0000,
	OPCUA_BADCONDITIONBRANCHALREADYACKED := 16#80CF0000,
	OPCUA_BADCONDITIONBRANCHALREADYCONFIRMED := 16#80D00000,
	OPCUA_BADCONDITIONALREADYSHELVED := 16#80D10000,
	OPCUA_BADCONDITIONNOTSHELVED := 16#80D20000,
	OPCUA_BADSHELVINGTIMEOUTOFRANGE := 16#80D30000,
	OPCUA_BADNODATA := 16#809B0000,
	OPCUA_BADBOUNDNOTFOUND := 16#80D70000,
	OPCUA_BADBOUNDNOTSUPPORTED := 16#80D80000,
	OPCUA_BADDATALOST := 16#809D0000,
	OPCUA_BADDATAUNAVAILABLE := 16#809E0000,
	OPCUA_BADENTRYEXISTS := 16#809F0000,
	OPCUA_BADNOENTRYEXISTS := 16#80A00000,
	OPCUA_BADTIMESTAMPNOTSUPPORTED := 16#80A10000,
	OPCUA_GOODENTRYINSERTED := 16#A20000,
	OPCUA_GOODENTRYREPLACED := 16#A30000,
	OPCUA_UNCERTAINDATASUBNORMAL := 16#40A40000,
	OPCUA_GOODNODATA := 16#A50000,
	OPCUA_GOODMOREDATA := 16#A60000,
	OPCUA_BADAGGREGATELISTMISMATCH := 16#80D40000,
	OPCUA_BADAGGREGATENOTSUPPORTED := 16#80D50000,
	OPCUA_BADAGGREGATEINVALIDINPUTS := 16#80D60000,
	OPCUA_BADAGGREGATECONFIGURATIONREJECTED := 16#80DA0000,
	OPCUA_GOODDATAIGNORED := 16#D90000,
	OPCUA_BADREQUESTNOTALLOWED := 16#80E40000,
	OPCUA_BADREQUESTNOTCOMPLETE := 16#81130000,
	OPCUA_GOODEDITED := 16#DC0000,
	OPCUA_GOODPOSTACTIONFAILED := 16#DD0000,
	OPCUA_UNCERTAINDOMINANTVALUECHANGED := 16#40DE0000,
	OPCUA_GOODDEPENDENTVALUECHANGED := 16#E00000,
	OPCUA_BADDOMINANTVALUECHANGED := 16#80E10000,
	OPCUA_UNCERTAINDEPENDENTVALUECHANGED := 16#40E20000,
	OPCUA_BADDEPENDENTVALUECHANGED := 16#80E30000,
	OPCUA_GOODCOMMUNICATIONEVENT := 16#A70000,
	OPCUA_GOODSHUTDOWNEVENT := 16#A80000,
	OPCUA_GOODCALLAGAIN := 16#A90000,
	OPCUA_GOODNONCRITICALTIMEOUT := 16#AA0000,
	OPCUA_BADINVALIDARGUMENT := 16#80AB0000,
	OPCUA_BADCONNECTIONREJECTED := 16#80AC0000,
	OPCUA_BADDISCONNECT := 16#80AD0000,
	OPCUA_BADCONNECTIONCLOSED := 16#80AE0000,
	OPCUA_BADINVALIDSTATE := 16#80AF0000,
	OPCUA_BADENDOFSTREAM := 16#80B00000,
	OPCUA_BADNODATAAVAILABLE := 16#80B10000,
	OPCUA_BADWAITINGFORRESPONSE := 16#80B20000,
	OPCUA_BADOPERATIONABANDONED := 16#80B30000,
	OPCUA_BADEXPECTEDSTREAMTOBLOCK := 16#80B40000,
	OPCUA_BADWOULDBLOCK := 16#80B50000,
	OPCUA_BADSYNTAXERROR := 16#80B60000,
	OPCUA_BADMAXCONNECTIONSREACHED := 16#80B70000
);
END_TYPE

(* ---- OPCUA_STATUSRESULT.dut ---- *)
TYPE OPCUA_STATUSRESULT :
STRUCT
	STATUSCODE : OpcUa_StatusCode;
	DIAGNOSTICINFO : OpcUa_DiagnosticInfo;
END_STRUCT
END_TYPE

(* ---- OPCUA_STRING.dut ---- *)
TYPE OPCUA_STRING :
STRUCT
	FLAGS : OpcUa_UInt16;
	ULENGTH : OpcUa_UInt32;
	STRCONTENT : POINTER TO OpcUa_CharA;
END_STRUCT
END_TYPE

(* ---- OPCUA_STRUCTUREDEFINITION.dut ---- *)
TYPE OPCUA_STRUCTUREDEFINITION :
STRUCT
	DEFAULTENCODINGID : OpcUa_NodeId;
	BASEDATATYPE : OpcUa_NodeId;
	STRUCTURETYPE : OpcUa_StructureType;
	NOOFFIELDS : OpcUa_Int32;
	FIELDS : POINTER TO OpcUa_StructureField;
END_STRUCT
END_TYPE

(* ---- OPCUA_STRUCTUREFIELD.dut ---- *)
TYPE OPCUA_STRUCTUREFIELD :
STRUCT
	NAME : OpcUa_String;
	DESCRIPTION : OpcUa_LocalizedText;
	DATATYPE : OpcUa_NodeId;
	VALUERANK : OpcUa_Int32;
	NOOFARRAYDIMENSIONS : OpcUa_Int32;
	ARRAYDIMENSIONS : POINTER TO OpcUa_UInt32;
	MAXSTRINGLENGTH : OpcUa_UInt32;
	ISOPTIONAL : OpcUa_Boolean;
END_STRUCT
END_TYPE

(* ---- OPCUA_STRUCTURETYPE.dut ---- *)
TYPE OPCUA_STRUCTURETYPE :
(
	OPCUA_STRUCTURETYPE_STRUCTURE := 0,
	OPCUA_STRUCTURETYPE_STRUCTUREWITHOPTIONALFIELDS := 1,
	OPCUA_STRUCTURETYPE_UNION := 2
);
END_TYPE

(* ---- OPCUA_SUBSCRIPTIONACKNOWLEDGEMENT.dut ---- *)
TYPE OPCUA_SUBSCRIPTIONACKNOWLEDGEMENT :
STRUCT
	SUBSCRIPTIONID : OpcUa_UInt32;
	SEQUENCENUMBER : OpcUa_UInt32;
END_STRUCT
END_TYPE

(* ---- OPCUA_SUBSCRIPTIONDIAGNOSTICSDATATYPE.dut ---- *)
TYPE OPCUA_SUBSCRIPTIONDIAGNOSTICSDATATYPE :
STRUCT
	SESSIONID : OpcUa_NodeId;
	SUBSCRIPTIONID : OpcUa_UInt32;
	PRIORITY : OpcUa_Byte;
	PUBLISHINGINTERVAL : OpcUa_Double;
	MAXKEEPALIVECOUNT : OpcUa_UInt32;
	MAXLIFETIMECOUNT : OpcUa_UInt32;
	MAXNOTIFICATIONSPERPUBLISH : OpcUa_UInt32;
	PUBLISHINGENABLED : OpcUa_Boolean;
	MODIFYCOUNT : OpcUa_UInt32;
	ENABLECOUNT : OpcUa_UInt32;
	DISABLECOUNT : OpcUa_UInt32;
	REPUBLISHREQUESTCOUNT : OpcUa_UInt32;
	REPUBLISHMESSAGEREQUESTCOUNT : OpcUa_UInt32;
	REPUBLISHMESSAGECOUNT : OpcUa_UInt32;
	TRANSFERREQUESTCOUNT : OpcUa_UInt32;
	TRANSFERREDTOALTCLIENTCOUNT : OpcUa_UInt32;
	TRANSFERREDTOSAMECLIENTCOUNT : OpcUa_UInt32;
	PUBLISHREQUESTCOUNT : OpcUa_UInt32;
	DATACHANGENOTIFICATIONSCOUNT : OpcUa_UInt32;
	EVENTNOTIFICATIONSCOUNT : OpcUa_UInt32;
	NOTIFICATIONSCOUNT : OpcUa_UInt32;
	LATEPUBLISHREQUESTCOUNT : OpcUa_UInt32;
	CURRENTKEEPALIVECOUNT : OpcUa_UInt32;
	CURRENTLIFETIMECOUNT : OpcUa_UInt32;
	UNACKNOWLEDGEDMESSAGECOUNT : OpcUa_UInt32;
	DISCARDEDMESSAGECOUNT : OpcUa_UInt32;
	MONITOREDITEMCOUNT : OpcUa_UInt32;
	DISABLEDMONITOREDITEMCOUNT : OpcUa_UInt32;
	MONITORINGQUEUEOVERFLOWCOUNT : OpcUa_UInt32;
	NEXTSEQUENCENUMBER : OpcUa_UInt32;
	EVENTQUEUEOVERFLOWCOUNT : OpcUa_UInt32;
END_STRUCT
END_TYPE

(* ---- OPCUA_TIMESTAMPSTORETURN.dut ---- *)
TYPE OPCUA_TIMESTAMPSTORETURN :
(
	OPCUA_TIMESTAMPSTORETURN_SOURCE := 0,
	OPCUA_TIMESTAMPSTORETURN_SERVER := 1,
	OPCUA_TIMESTAMPSTORETURN_BOTH := 2,
	OPCUA_TIMESTAMPSTORETURN_NEITHER := 3,
	OPCUA_TIMESTAMPSTORETURN_INVALID := 4
);
END_TYPE

(* ---- OPCUA_TIMEZONEDATATYPE.dut ---- *)
TYPE OPCUA_TIMEZONEDATATYPE :
STRUCT
	OFFSET : OpcUa_Int16;
	DAYLIGHTSAVINGINOFFSET : OpcUa_Boolean;
END_STRUCT
END_TYPE

(* ---- OPCUA_TRANSFERRESULT.dut ---- *)
TYPE OPCUA_TRANSFERRESULT :
STRUCT
	STATUSCODE : OpcUa_StatusCode;
	NOOFAVAILABLESEQUENCENUMBERS : OpcUa_Int32;
	AVAILABLESEQUENCENUMBERS : POINTER TO OpcUa_UInt32;
END_STRUCT
END_TYPE

(* ---- OPCUA_TRANSFERSUBSCRIPTIONSREQUEST.dut ---- *)
TYPE OPCUA_TRANSFERSUBSCRIPTIONSREQUEST :
STRUCT
	REQUESTHEADER : OpcUa_RequestHeader;
	NOOFSUBSCRIPTIONIDS : OpcUa_Int32;
	SUBSCRIPTIONIDS : POINTER TO OpcUa_UInt32;
	SENDINITIALVALUES : OpcUa_Boolean;
END_STRUCT
END_TYPE

(* ---- OPCUA_TRANSFERSUBSCRIPTIONSRESPONSE.dut ---- *)
TYPE OPCUA_TRANSFERSUBSCRIPTIONSRESPONSE :
STRUCT
	RESPONSEHEADER : OpcUa_ResponseHeader;
	NOOFRESULTS : OpcUa_Int32;
	RESULTS : POINTER TO OpcUa_TransferResult;
	NOOFDIAGNOSTICINFOS : OpcUa_Int32;
	DIAGNOSTICINFOS : POINTER TO OpcUa_DiagnosticInfo;
END_STRUCT
END_TYPE

(* ---- OPCUA_TRANSLATEBROWSEPATHSTONODEIDSREQUEST.dut ---- *)
TYPE OPCUA_TRANSLATEBROWSEPATHSTONODEIDSREQUEST :
STRUCT
	REQUESTHEADER : OpcUa_RequestHeader;
	NOOFBROWSEPATHS : OpcUa_Int32;
	BROWSEPATHS : POINTER TO OpcUa_BrowsePath;
END_STRUCT
END_TYPE

(* ---- OPCUA_TRANSLATEBROWSEPATHSTONODEIDSRESPONSE.dut ---- *)
TYPE OPCUA_TRANSLATEBROWSEPATHSTONODEIDSRESPONSE :
STRUCT
	RESPONSEHEADER : OpcUa_ResponseHeader;
	NOOFRESULTS : OpcUa_Int32;
	RESULTS : POINTER TO OpcUa_BrowsePathResult;
	NOOFDIAGNOSTICINFOS : OpcUa_Int32;
	DIAGNOSTICINFOS : POINTER TO OpcUa_DiagnosticInfo;
END_STRUCT
END_TYPE

(* ---- OPCUA_UINT.dut ---- *)
TYPE OPCUA_UINT : UDINT;
END_TYPE

(* ---- OPCUA_UINT16.dut ---- *)
TYPE OPCUA_UINT16 : UINT;
END_TYPE

(* ---- OPCUA_UINT32.dut ---- *)
TYPE OPCUA_UINT32 : UDINT;
END_TYPE

(* ---- OPCUA_UINT64.dut ---- *)
TYPE OPCUA_UINT64 : ULINT;
END_TYPE

(* ---- OPCUA_UNREGISTERNODESREQUEST.dut ---- *)
TYPE OPCUA_UNREGISTERNODESREQUEST :
STRUCT
	REQUESTHEADER : OpcUa_RequestHeader;
	NOOFNODESTOUNREGISTER : OpcUa_Int32;
	NODESTOUNREGISTER : POINTER TO OpcUa_NodeId;
END_STRUCT
END_TYPE

(* ---- OPCUA_UNREGISTERNODESRESPONSE.dut ---- *)
TYPE OPCUA_UNREGISTERNODESRESPONSE :
STRUCT
	RESPONSEHEADER : OpcUa_ResponseHeader;
END_STRUCT
END_TYPE

(* ---- OPCUA_UPDATEDATADETAILS.dut ---- *)
TYPE OPCUA_UPDATEDATADETAILS :
STRUCT
	NODEID : OpcUa_NodeId;
	PERFORMINSERTREPLACE : OpcUa_PerformUpdateType;
	NOOFUPDATEVALUES : OpcUa_Int32;
	UPDATEVALUES : POINTER TO OpcUa_DataValue;
END_STRUCT
END_TYPE

(* ---- OPCUA_UPDATEEVENTDETAILS.dut ---- *)
TYPE OPCUA_UPDATEEVENTDETAILS :
STRUCT
	NODEID : OpcUa_NodeId;
	PERFORMINSERTREPLACE : OpcUa_PerformUpdateType;
	FILTER : OpcUa_EventFilter;
	NOOFEVENTDATA : OpcUa_Int32;
	EVENTDATA : POINTER TO OpcUa_HistoryEventFieldList;
END_STRUCT
END_TYPE

(* ---- OPCUA_UPDATESTRUCTUREDATADETAILS.dut ---- *)
TYPE OPCUA_UPDATESTRUCTUREDATADETAILS :
STRUCT
	NODEID : OpcUa_NodeId;
	PERFORMINSERTREPLACE : OpcUa_PerformUpdateType;
	NOOFUPDATEVALUES : OpcUa_Int32;
	UPDATEVALUES : POINTER TO OpcUa_DataValue;
END_STRUCT
END_TYPE

(* ---- OPCUA_USERIDENTITYTOKEN.dut ---- *)
TYPE OPCUA_USERIDENTITYTOKEN :
STRUCT
	POLICYID : OpcUa_String;
END_STRUCT
END_TYPE

(* ---- OPCUA_USERNAMEIDENTITYTOKEN.dut ---- *)
TYPE OPCUA_USERNAMEIDENTITYTOKEN :
STRUCT
	POLICYID : OpcUa_String;
	USERNAME : OpcUa_String;
	PASSWORD : OpcUa_ByteString;
	ENCRYPTIONALGORITHM : OpcUa_String;
END_STRUCT
END_TYPE

(* ---- OPCUA_USERTOKENPOLICY.dut ---- *)
TYPE OPCUA_USERTOKENPOLICY :
STRUCT
	POLICYID : OpcUa_String;
	TOKENTYPE : OpcUa_UserTokenType;
	ISSUEDTOKENTYPE : OpcUa_String;
	ISSUERENDPOINTURL : OpcUa_String;
	SECURITYPOLICYURI : OpcUa_String;
END_STRUCT
END_TYPE

(* ---- OPCUA_USERTOKENTYPE.dut ---- *)
TYPE OPCUA_USERTOKENTYPE :
(
	OPCUA_USERTOKENTYPE_ANONYMOUS := 0,
	OPCUA_USERTOKENTYPE_USERNAME := 1,
	OPCUA_USERTOKENTYPE_CERTIFICATE := 2,
	OPCUA_USERTOKENTYPE_ISSUEDTOKEN := 3
);
END_TYPE

(* ---- OPCUA_VARIABLEATTRIBUTES.dut ---- *)
TYPE OPCUA_VARIABLEATTRIBUTES :
STRUCT
	SPECIFIEDATTRIBUTES : OpcUa_UInt32;
	DISPLAYNAME : OpcUa_LocalizedText;
	DESCRIPTION : OpcUa_LocalizedText;
	WRITEMASK : OpcUa_UInt32;
	USERWRITEMASK : OpcUa_UInt32;
	VALUE : OpcUa_Variant;
	DATATYPE : OpcUa_NodeId;
	VALUERANK : OpcUa_Int32;
	NOOFARRAYDIMENSIONS : OpcUa_Int32;
	ARRAYDIMENSIONS : POINTER TO OpcUa_UInt32;
	ACCESSLEVEL : OpcUa_Byte;
	USERACCESSLEVEL : OpcUa_Byte;
	MINIMUMSAMPLINGINTERVAL : OpcUa_Double;
	HISTORIZING : OpcUa_Boolean;
END_STRUCT
END_TYPE

(* ---- OPCUA_VARIABLETYPEATTRIBUTES.dut ---- *)
TYPE OPCUA_VARIABLETYPEATTRIBUTES :
STRUCT
	SPECIFIEDATTRIBUTES : OpcUa_UInt32;
	DISPLAYNAME : OpcUa_LocalizedText;
	DESCRIPTION : OpcUa_LocalizedText;
	WRITEMASK : OpcUa_UInt32;
	USERWRITEMASK : OpcUa_UInt32;
	VALUE : OpcUa_Variant;
	DATATYPE : OpcUa_NodeId;
	VALUERANK : OpcUa_Int32;
	NOOFARRAYDIMENSIONS : OpcUa_Int32;
	ARRAYDIMENSIONS : POINTER TO OpcUa_UInt32;
	ISABSTRACT : OpcUa_Boolean;
END_STRUCT
END_TYPE

(* ---- OPCUA_VARIANT.dut ---- *)
TYPE OPCUA_VARIANT :
STRUCT
	DATATYPE : OpcUa_Byte;
	ARRAYTYPE : OpcUa_Byte;
	RESERVED : OpcUa_UInt16;
	VALUE : OpcUa_VariantUnion;
END_STRUCT
END_TYPE

(* ---- OPCUA_VARIANTARRAYTYPE.dut ---- *)
TYPE OPCUA_VARIANTARRAYTYPE :
(
	OPCUA_VARIANTARRAYTYPE_SCALAR := 0,
	OPCUA_VARIANTARRAYTYPE_ARRAY := 1,
	OPCUA_VARIANTARRAYTYPE_MATRIX := 2
);
END_TYPE

(* ---- OPCUA_VARIANTARRAYUNION.dut ---- *)
TYPE OPCUA_VARIANTARRAYUNION :
UNION
	ARRAY_CDS : POINTER TO BYTE;
	BOOLEANARRAY : POINTER TO OpcUa_Boolean;
	SBYTEARRAY : POINTER TO OpcUa_SByte;
	BYTEARRAY : POINTER TO OpcUa_Byte;
	INT16ARRAY : POINTER TO OpcUa_Int16;
	UINT16ARRAY : POINTER TO OpcUa_UInt16;
	INT32ARRAY : POINTER TO OpcUa_Int32;
	UINT32ARRAY : POINTER TO OpcUa_UInt32;
	INT64ARRAY : POINTER TO OpcUa_Int64;
	UINT64ARRAY : POINTER TO OpcUa_UInt64;
	FLOATARRAY : POINTER TO OpcUa_Float;
	DOUBLEARRAY : POINTER TO OpcUa_Double;
	STRINGARRAY : POINTER TO OpcUa_String;
	DATETIMEARRAY : POINTER TO OpcUa_DateTime;
	GUIDARRAY : POINTER TO OpcUa_Guid;
	BYTESTRINGARRAY : POINTER TO OpcUa_ByteString;
	XMLELEMENTARRAY : POINTER TO OpcUa_ByteString;
	NODEIDARRAY : POINTER TO OpcUa_NodeId;
	EXPANDEDNODEIDARRAY : POINTER TO OpcUa_ExpandedNodeId;
	STATUSCODEARRAY : POINTER TO OpcUa_StatusCode;
	QUALIFIEDNAMEARRAY : POINTER TO OpcUa_QualifiedName;
	LOCALIZEDTEXTARRAY : POINTER TO OpcUa_LocalizedText;
	EXTENSIONOBJECTARRAY : POINTER TO OpcUa_ExtensionObject;
	DATAVALUEARRAY : POINTER TO BYTE;
	VARIANTARRAY : POINTER TO OpcUa_Variant;
END_UNION
END_TYPE

(* ---- OPCUA_VARIANTARRAYVALUE.dut ---- *)
TYPE OPCUA_VARIANTARRAYVALUE :
STRUCT
	LENGTH : OpcUa_Int32;
	VALUE : OpcUa_VariantArrayUnion;
END_STRUCT
END_TYPE

(* ---- OPCUA_VARIANTMATRIXVALUE.dut ---- *)
TYPE OPCUA_VARIANTMATRIXVALUE :
STRUCT
	NOOFDIMENSIONS : OpcUa_Int32;
	DIMENSIONS : POINTER TO OpcUa_Int32;
	VALUE : OpcUa_VariantArrayUnion;
END_STRUCT
END_TYPE

(* ---- OPCUA_VARIANTUNION.dut ---- *)
TYPE OPCUA_VARIANTUNION :
UNION
	BOOLEAN : OpcUa_Boolean;
	SBYTE : OpcUa_SByte;
	BYTE_CDS : OpcUa_Byte;
	INT16 : OpcUa_Int16;
	UINT16 : OpcUa_UInt16;
	INT32 : OpcUa_Int32;
	UINT32 : OpcUa_UInt32;
	INT64 : OpcUa_Int64;
	UINT64 : OpcUa_UInt64;
	FLOAT : OpcUa_Float;
	DOUBLE : OpcUa_Double;
	DATETIME : OpcUa_DateTime;
	STRING_CDS : OpcUa_String;
	GUID : POINTER TO OpcUa_Guid;
	BYTESTRING : OpcUa_ByteString;
	XMLELEMENT : OpcUa_ByteString;
	NODEID : POINTER TO OpcUa_NodeId;
	EXPANDEDNODEID : POINTER TO OpcUa_ExpandedNodeId;
	STATUSCODE : OpcUa_StatusCode;
	QUALIFIEDNAME : POINTER TO OpcUa_QualifiedName;
	LOCALIZEDTEXT : POINTER TO OpcUa_LocalizedText;
	EXTENSIONOBJECT : POINTER TO OpcUa_ExtensionObject;
	DATAVALUE : POINTER TO BYTE;
	ARRAY_CDS : OpcUa_VariantArrayValue;
	MATRIX : OpcUa_VariantMatrixValue;
END_UNION
END_TYPE

(* ---- OPCUA_VIEWATTRIBUTES.dut ---- *)
TYPE OPCUA_VIEWATTRIBUTES :
STRUCT
	SPECIFIEDATTRIBUTES : OpcUa_UInt32;
	DISPLAYNAME : OpcUa_LocalizedText;
	DESCRIPTION : OpcUa_LocalizedText;
	WRITEMASK : OpcUa_UInt32;
	USERWRITEMASK : OpcUa_UInt32;
	CONTAINSNOLOOPS : OpcUa_Boolean;
	EVENTNOTIFIER : OpcUa_Byte;
END_STRUCT
END_TYPE

(* ---- OPCUA_VIEWDESCRIPTION.dut ---- *)
TYPE OPCUA_VIEWDESCRIPTION :
STRUCT
	VIEWID : OpcUa_NodeId;
	TIMESTAMP : OpcUa_DateTime;
	VIEWVERSION : OpcUa_UInt32;
END_STRUCT
END_TYPE

(* ---- OPCUA_WRITEREQUEST.dut ---- *)
TYPE OPCUA_WRITEREQUEST :
STRUCT
	REQUESTHEADER : OpcUa_RequestHeader;
	NOOFNODESTOWRITE : OpcUa_Int32;
	NODESTOWRITE : POINTER TO OpcUa_WriteValue;
END_STRUCT
END_TYPE

(* ---- OPCUA_WRITERESPONSE.dut ---- *)
TYPE OPCUA_WRITERESPONSE :
STRUCT
	RESPONSEHEADER : OpcUa_ResponseHeader;
	NOOFRESULTS : OpcUa_Int32;
	RESULTS : POINTER TO OpcUa_StatusCode;
	NOOFDIAGNOSTICINFOS : OpcUa_Int32;
	DIAGNOSTICINFOS : POINTER TO OpcUa_DiagnosticInfo;
END_STRUCT
END_TYPE

(* ---- OPCUA_WRITEVALUE.dut ---- *)
TYPE OPCUA_WRITEVALUE :
STRUCT
	NODEID : OpcUa_NodeId;
	ATTRIBUTEID : OpcUa_UInt32;
	INDEXRANGE : OpcUa_String;
	VALUE : OpcUa_DataValue;
END_STRUCT
END_TYPE

(* ---- OPCUA_X509IDENTITYTOKEN.dut ---- *)
TYPE OPCUA_X509IDENTITYTOKEN :
STRUCT
	POLICYID : OpcUa_String;
	CERTIFICATEDATA : OpcUa_ByteString;
END_STRUCT
END_TYPE

(* ---- OPCUA_XVTYPE.dut ---- *)
TYPE OPCUA_XVTYPE :
STRUCT
	X : OpcUa_Double;
	VALUE : OpcUa_Float;
END_STRUCT
END_TYPE
